// TIA Portal V19 export
FUNCTION_BLOCK "TYPIC_C701_IF_VAT_BUF"   // FB70, FBD
TITLE = TYPIC_C701_IF_VAT_BUF: Buffervat warm water
{ S7_Optimized_Access := 'TRUE' }
AUTHOR : OCOTECH
FAMILY : Typical
NAME : C701.714
// Logisch Object Besturing: C701.714
// 
// De interne functie Buffervat verzorgt de interne besturing, bewaking en fysieke aansturing van het buffervat behorend tot de klimaatinstallatie.
// stored: MemoryReserve 10, SetENOAutomatically false
   VAR_INPUT
      STU_IF_VAT_BUF { ExternalAccessible := 'False'; ExternalVisible := 'False'; ExternalWritable := 'False'} : Bool;   // Sturing van de interne functie klimaatregeling (IF), vrijgave door storing warmtepomp
      IN_STO { ExternalAccessible := 'False'; ExternalVisible := 'False'; ExternalWritable := 'False'} : Bool;   // Storing elektrisch weerstand
      IN_TME_MWA_INV { ExternalAccessible := 'False'; ExternalVisible := 'False'; ExternalWritable := 'False'} : Real;   // Temperatuurmeting warmwater in vertrek
      IN_TME_MWA_UITV { ExternalAccessible := 'False'; ExternalVisible := 'False'; ExternalWritable := 'False'} : Real;   // Temperatuurmeting warmwater uit vertrek
      IN_TME3_MWA { ExternalAccessible := 'False'; ExternalVisible := 'False'; ExternalWritable := 'False'} : Real;   // Temperatuurmeting warmwater in retour
      IN_TME4_MWA { ExternalAccessible := 'False'; ExternalVisible := 'False'; ExternalWritable := 'False'} : Real;   // Temperatuurmeting warmwater uit retour
   END_VAR
   VAR_OUTPUT
      VAR_IF_VAT_BUF { ExternalAccessible := 'False'; ExternalVisible := 'False'; ExternalWritable := 'False'} : "C701_VAR_IF_VAT_BUF_TYPIC";   // Struct met alle variabelen naar bovenliggende functies
      OUT_AAN { ExternalAccessible := 'False'; ExternalVisible := 'False'; ExternalWritable := 'False'} : Bool;   // Sturing elektrische weerstand (1 = Aan)
   END_VAR
   VAR
      STO { ExternalWritable := 'False'} : Struct   // Storingen
         A001 : Bool;   // Fout temperatuurmeting in vertrek
         A002 : Bool;   // Fout temperatuurmeting uit vertrek
         A003 : Bool;   // Fout temperatuurmeting in retour
         A004 : Bool;   // Fout temperatuurmeting uit retour
      END_STRUCT;
      VAR { ExternalWritable := 'False'} : Struct   // Variabelen
         TME_IN_VERTREK : Real;   // Temperatuurmeting in
         TME_UIT_VERTREK : Real;   // Temperatuurmeting uit
         TME_IN_RETOUR : Real;   // Temperatuurmeting in
         TME_UIT_RETOUR : Real;   // Temperatuurmeting uit
         TME_SWA : Real;   // Setpunt temperatuur buffervat
      END_STRUCT;
   END_VAR
BEGIN

REGION Network 1: START
END_REGION

REGION Network 2: +++ Metingen +++
   // inlezen van ingaande en uitgaande temperatuur.
END_REGION

REGION Network 3: +++ Storingen en meldingen +++
   // aanmaken van storingen en meldingen.
END_REGION

REGION Network 4: Storing A001: Fout temperatuurmeting in vertrek
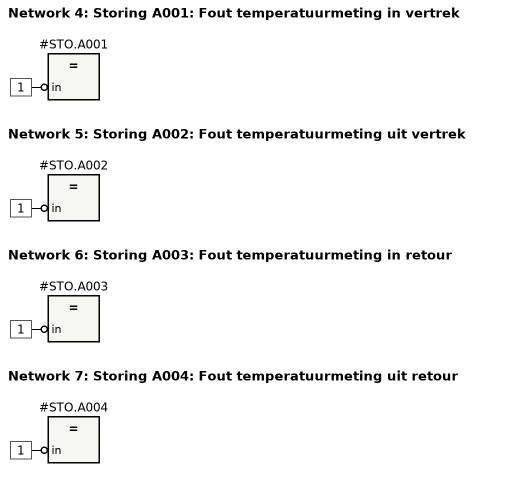
   #STO.A001 := NOT 1;
END_REGION

REGION Network 5: Storing A002: Fout temperatuurmeting uit vertrek
   #STO.A002 := NOT 1;
END_REGION

REGION Network 6: Storing A003: Fout temperatuurmeting in retour
   #STO.A003 := NOT 1;
END_REGION

REGION Network 7: Storing A004: Fout temperatuurmeting uit retour
   #STO.A004 := NOT 1;
END_REGION

REGION Network 8: +++ Sturingen +++
   // bij storing warmtepomp wordt elektrische weerstand vrijgegeven en geregeld naar setpunt.
END_REGION

REGION Network 9 (SCL): EINDE
   // Variabelen van intern scada rakvlak naar outputs copieren
   #VAR_IF_VAT_BUF.STO := #STO;
END_REGION
END_FUNCTION_BLOCK
